TEXTLIST TL_E_MESSAGETYPE
  0 = 'eMessageEmpty'
  1 = 'eMessageError'
  2 = 'eMessageWarning'
  3 = 'eMessageInfo'
  4 = 'eMessageVerbose'
   = ''
END_TEXTLIST

(* stored: Version 1.1.0.1
   TextList TL_E_MESSAGETYPE: Id {e1d37e76-e189-4358-bf6a-24e92d83fe6e} *)
